// Mitsubishi GX Works2 project: 타이머응용2   PLC: Q02/Q02H

PROGRAM MAIN
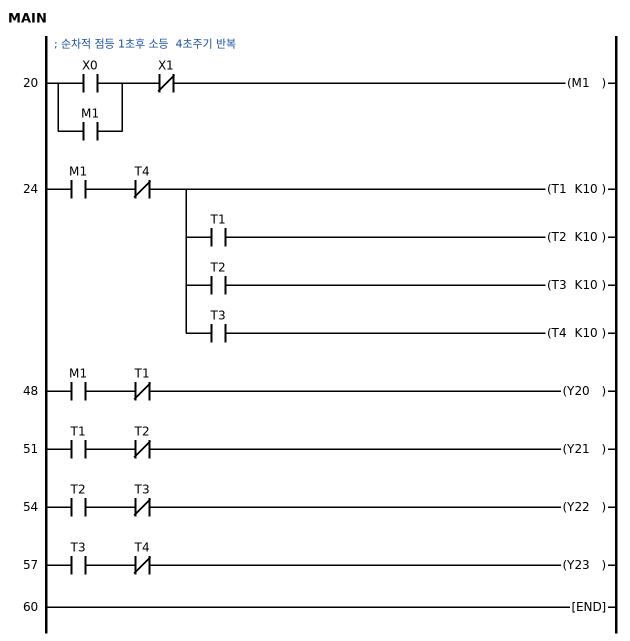
; 순차적 점등 1초후 소등  4초주기 반복
20    LD      X0
      OR      M1
      ANI     X1
      OUT     M1
24    LD      M1
      ANI     T4
      OUT     T1 K10
      MPS
      AND     T1
      OUT     T2 K10
      MRD
      AND     T2
      OUT     T3 K10
      MPP
      AND     T3
      OUT     T4 K10
48    LD      M1
      ANI     T1
      OUT     Y20
51    LD      T1
      ANI     T2
      OUT     Y21
54    LD      T2
      ANI     T3
      OUT     Y22
57    LD      T3
      ANI     T4
      OUT     Y23
60    END
END_PROGRAM
